{attribute 'qualified_only'}
VAR_GLOBAL
END_VAR

(* stored: Version 1.1.0.1, ProductVersion 3.1.4022.7
   GVL GVL_03_Delay_Step_Motor: Id {d273038b-d95d-4f9b-a2f3-36a289c54641} *)
